TYPE ST_ClampStationOutImm :
STRUCT
    Clamped   : BOOL;
    Unclamped : BOOL;
    Diagnostic: ST_Diagnostic;
END_STRUCT
END_TYPE

(* stored: Version 1.1.0.1, ProductVersion 3.1.4024.12
   DUT ST_ClampStationOutImm: Id {a27f0545-9ce6-4f07-b175-0395cdedb112} *)
